TYPE ST_ValvePos :
STRUCT
	rCylinderValve : REAL;
END_STRUCT
END_TYPE

(* stored: Version 1.1.0.1
   DUT ST_ValvePos: Id {4b39be98-fe42-4c0f-bfcb-c5097dfd34e9} *)
